(* IEC 61131-3 sources: com.logicals.lc3.webinar/usRTS_RPMControl_iSOC/src_FB_LIB_SAFE/Convert/BYTE, 4 files *)

(* ---- wBYTE_TO_DWORD.iecst ---- *)
NAMESPACE logicals.web.standard
NAMESPACE convert

/*
 * Function block wrapper for IEC 61131-3 TO_DWORD<br>
 * IN =  input value (BYTE)<br>
 * OUT = IN (DWORD)<br>
 */
FUNCTION_BLOCK wBYTE_TO_DWORD
	{ vNameAlignment:="center"; altName:="BYTE_TO_DWORD"; bgColor:="DodgerBlue"; width:=140; hideIONames; }
	VAR_INPUT
		IN : BYTE;
	END_VAR
	VAR_OUTPUT
		OUT: DWORD;
	END_VAR

	OUT := TO_DWORD(IN:=IN, ENO=>ENO);
END_FUNCTION_BLOCK

END_NAMESPACE
END_NAMESPACE

(* ---- wBYTE_TO_LWORD.iecst ---- *)
NAMESPACE logicals.web.standard
NAMESPACE convert

/*
 * Function block wrapper for IEC 61131-3 TO_LWORD<br>
 * IN =  input value (BYTE)<br>
 * OUT = IN (LWORD)<br>
 */
FUNCTION_BLOCK wBYTE_TO_LWORD
	{ vNameAlignment:="center"; altName:="BYTE_TO_LWORD"; bgColor:="DodgerBlue"; width:=140; hideIONames; }
	VAR_INPUT
		IN : BYTE;
	END_VAR
	VAR_OUTPUT
		OUT: LWORD;
	END_VAR

	OUT := TO_LWORD(IN:=IN, ENO=>ENO);
END_FUNCTION_BLOCK

END_NAMESPACE
END_NAMESPACE

(* ---- wBYTE_TO_USINT.iecst ---- *)
NAMESPACE logicals.web.standard
NAMESPACE convert

/*
 * Function block wrapper for IEC 61131-3 TO_USINT<br>
 * IN =  input value (BYTE)<br>
 * OUT = IN (USINT)<br>
 */
FUNCTION_BLOCK wBYTE_TO_USINT
	{ vNameAlignment:="center"; altName:="BYTE_TO_USINT"; bgColor:="Plum"; width:=140; hideIONames; }
	VAR_INPUT
		IN : BYTE;
	END_VAR
	VAR_OUTPUT
		OUT: USINT;
	END_VAR

	OUT := TO_USINT(IN:=IN, ENO=>ENO);
END_FUNCTION_BLOCK

END_NAMESPACE
END_NAMESPACE

(* ---- wBYTE_TO_WORD.iecst ---- *)
NAMESPACE logicals.web.standard
NAMESPACE convert

/*
 * Function block wrapper for IEC 61131-3 TO_WORD<br>
 * IN =  input value (BYTE)<br>
 * OUT = IN (WORD)<br>
 */
FUNCTION_BLOCK wBYTE_TO_WORD
	{ vNameAlignment:="center"; altName:="BYTE_TO_WORD"; bgColor:="DodgerBlue"; width:=140; hideIONames; }
	VAR_INPUT
		IN : BYTE;
	END_VAR
	VAR_OUTPUT
		OUT: WORD;
	END_VAR

	OUT := TO_WORD(IN:=IN, ENO=>ENO);
END_FUNCTION_BLOCK

END_NAMESPACE
END_NAMESPACE
